{attribute 'linkalways'} 
{attribute 'no_explicit_call' := 'This FB is a CLASS and must be accessed using methods or properties'}
{attribute 'enable_dynamic_creation'}
FUNCTION_BLOCK Node_F_VN_DrawKeypoints EXTENDS VisionNode
VAR
    ipSrcImage : _ITcVnImage;
    ipKeyPoints : _ITcVnContainer;
    ipDestImage : _ITcVnImage;
    hrPrev : _HRESULT(S_OK);
	hresult : _HRESULT(S_OK);
END_VAR

METHOD PUBLIC  Clone : I_Node
VAR
	pNode : POINTER TO Node_F_VN_DrawKeypoints
;
END_VAR
pNode := __NEW(Node_F_VN_DrawKeypoints);
Clone := pNode^;
END_METHOD

METHOD FB_init : BOOL
VAR_INPUT
	bInitRetains : BOOL; // if TRUE, the retain variables are initialized (warm start / cold start)
	bInCopyCode : BOOL;  // if TRUE, the instance afterwards gets moved into the copy code (online change)
END_VAR
AddInput('ipSrcImage', ipSrcImage);
AddInput('ipKeyPoints', ipKeyPoints);
AddInput('hrPrev', hrPrev);
AddOutput('ipDestImage', ipDestImage);
AddOutput('hresult',hresult);
END_METHOD

METHOD PROTECTED OnExecute
hresult.Value := F_VN_DrawKeypoints(
    ipSrcImage := ipSrcImage.Value,
    ipKeyPoints := ipKeyPoints.Value,
	ipDestImage := ipDestImage.Value,
	hrPrev:= hrPrev.Value);
END_METHOD

METHOD PUBLIC PreExecutionCheck
VAR_INPUT
	Check : I_PreExecutionChecks;
END_VAR
Check.IsTrue(ipSrcImage.IsValid, 'ipSrcImage must contain an image');
Check.IsTrue(ipKeyPoints.IsType(TC_GLOBAL_CONST_LIST.ContainerType_Vector_TcVnKeyPoint), 'ipKeyPoints contains incorrect type');
END_METHOD

END_FUNCTION_BLOCK

(* stored: Version 1.1.0.1, ProductVersion 3.1.4026.13
   POU Node_F_VN_DrawKeypoints: Id {cae2e8c7-63bf-0210-3f10-6763906c87d8}, SpecialFunc None
   Folder Constructor: Id {485033ca-593c-0047-0bf8-9fff33975583}
   Method Clone: Id {8fc5e0e7-7a09-0b34-1a7d-005dd8c8a947}
   Method FB_init: Id {c33fc327-87ef-0f78-37a9-677755203b92}
   Method OnExecute: Id {ad4f82e6-b83f-0ab2-24cf-d3c90144f96b}
   Method PreExecutionCheck: Id {bdb67ac1-6cb7-0f62-123a-e37c0efe5cd4} *)
